// Brief: Panel Ready
FUNCTION_BLOCK PUBLIC FB_SlaveCtrlPanelReady EXTENDS FB_SlaveArmCtrlBase
VAR_INPUT
END_VAR
VAR_OUTPUT
END_VAR
VAR
END_VAR

// override this function in each exact controller
// NOTICE: set joint control mode here, and do some initialization if needed
METHOD PUBLIC init : BOOL
VAR_IN_OUT CONSTANT
	i_slaveArm	:FB_SlaveArm;
END_VAR
VAR_IN_OUT 
	r_slaveArmCtrlCmd :ST_SlaveArmCtrlCmds;
END_VAR
//init
SUPER^.Init(i_slaveArm,r_slaveArmCtrlCmd);

//update the control mode ---1028
m_jntOPMode := g_slaveAllPosMode;
m_jntOPMode[1]:=DriverOPMode_PosTrq;
m_jntOPMode[2]:=DriverOPMode_PosTrq;

copyCmds(r_slaveArmCtrlCmd);
END_METHOD

END_FUNCTION_BLOCK

(* stored: Version 1.1.0.1, ProductVersion 3.1.4024.11
   POU FB_SlaveCtrlPanelReady: Id {f4ef749e-f294-45ac-8079-35edcc11796e}, SpecialFunc None
   Method init: Id {45b56ef0-3ee7-49ce-be9a-eb6606411d59} *)
